PROGRAM PRG_SL2K0_POWER
VAR
    {attribute 'pytmc' := '
        pv: SL2K0:POWER
        io: io
    '}
    {attribute 'TcLinkTo' := '.RTD_South_1.iRaw := TIIB[SL2K0-EL3202-E8]^RTD Inputs Channel 1^Value;
                              .RTD_South_1.bError := TIIB[SL2K0-EL3202-E8]^RTD Inputs Channel 1^Status^Error;
                              .RTD_South_1.bUnderrange := TIIB[SL2K0-EL3202-E8]^RTD Inputs Channel 1^Status^Underrange;
                              .RTD_South_1.bOverrange := TIIB[SL2K0-EL3202-E8]^RTD Inputs Channel 1^Status^Overrange;
                              .RTD_South_2.iRaw := TIIB[SL2K0-EL3202-E8]^RTD Inputs Channel 2^Value;
                              .RTD_South_2.bError := TIIB[SL2K0-EL3202-E8]^RTD Inputs Channel 2^Status^Error;
                              .RTD_South_2.bUnderrange := TIIB[SL2K0-EL3202-E8]^RTD Inputs Channel 2^Status^Underrange;
                              .RTD_South_2.bOverrange := TIIB[SL2K0-EL3202-E8]^RTD Inputs Channel 2^Status^Overrange;
                              .RTD_TOP_1.iRaw := TIIB[SL2K0-EL3202-E9]^RTD Inputs Channel 1^Value;
                              .RTD_TOP_1.bError := TIIB[SL2K0-EL3202-E9]^RTD Inputs Channel 1^Status^Error;
                              .RTD_TOP_1.bUnderrange := TIIB[SL2K0-EL3202-E9]^RTD Inputs Channel 1^Status^Underrange;
                              .RTD_TOP_1.bOverrange := TIIB[SL2K0-EL3202-E9]^RTD Inputs Channel 1^Status^Overrange;
                              .RTD_TOP_2.iRaw := TIIB[SL2K0-EL3202-E9]^RTD Inputs Channel 2^Value;
                              .RTD_TOP_2.bError := TIIB[SL2K0-EL3202-E9]^RTD Inputs Channel 2^Status^Error;
                              .RTD_TOP_2.bUnderrange := TIIB[SL2K0-EL3202-E9]^RTD Inputs Channel 2^Status^Underrange;
                              .RTD_TOP_2.bOverrange := TIIB[SL2K0-EL3202-E9]^RTD Inputs Channel 2^Status^Overrange;
                              .RTD_North_1.iRaw := TIIB[SL2K0-EL3202-E10]^RTD Inputs Channel 1^Value;
                              .RTD_North_1.bError := TIIB[SL2K0-EL3202-E10]^RTD Inputs Channel 1^Status^Error;
                              .RTD_North_1.bUnderrange := TIIB[SL2K0-EL3202-E10]^RTD Inputs Channel 1^Status^Underrange;
                              .RTD_North_1.bOverrange := TIIB[SL2K0-EL3202-E10]^RTD Inputs Channel 1^Status^Overrange;
                              .RTD_North_2.iRaw := TIIB[SL2K0-EL3202-E10]^RTD Inputs Channel 2^Value;
                              .RTD_North_2.bError := TIIB[SL2K0-EL3202-E10]^RTD Inputs Channel 2^Status^Error;
                              .RTD_North_2.bUnderrange := TIIB[SL2K0-EL3202-E10]^RTD Inputs Channel 2^Status^Underrange;
                              .RTD_North_2.bOverrange := TIIB[SL2K0-EL3202-E10]^RTD Inputs Channel 2^Status^Overrange;
                              .RTD_Bottom_1.iRaw := TIIB[SL2K0-EL3202-E10]^RTD Inputs Channel 1^Value;
                              .RTD_Bottom_1.bError := TIIB[SL2K0-EL3202-E10]^RTD Inputs Channel 1^Status^Error;
                              .RTD_Bottom_1.bUnderrange := TIIB[SL2K0-EL3202-E11]^RTD Inputs Channel 1^Status^Underrange;
                              .RTD_Bottom_1.bOverrange := TIIB[SL2K0-EL3202-E11]^RTD Inputs Channel 1^Status^Overrange;
                              .RTD_Bottom_2.iRaw := TIIB[SL2K0-EL3202-E11]^RTD Inputs Channel 2^Value;
                              .RTD_Bottom_2.bError := TIIB[SL2K0-EL3202-E11]^RTD Inputs Channel 2^Status^Error;
                              .RTD_Bottom_2.bUnderrange := TIIB[SL2K0-EL3202-E11]^RTD Inputs Channel 2^Status^Underrange;
                              .RTD_Bottom_2.bOverrange := TIIB[SL2K0-EL3202-E11]^RTD Inputs Channel 2^Status^Overrange'}
    fbSL2K0: FB_SLITS_POWER;
//GET PMP Move Ok bit
// Default True until it is properly linked to PMPS bit
    bMoveOk:BOOL :=TRUE;
    {attribute 'pytmc' := '
    pv: SL2K0:POWER:GO;
    io: io;
    field: ZNAM False;
    field: ONAM True;
    '}
    bExecuteMotion:BOOL ;
    //for testing purposes only. comment-out/delete once done.
    mcPower : ARRAY [1..4] OF MC_POWER;
END_VAR


fbSL2K0.bMoveOk := bMoveOk;

fbSL2K0(stTopBlade:=  Main.M22,
        stBottomBlade:= Main.M23,
        stNorthBlade:=  Main.M24,
        stSouthBlade:=  Main.M25,
        bExecuteMotion:=bExecuteMotion);


//for testing purposes only. comment-out/delete once done.
(*mcPower[1](axis:=Main.M22.Axis, Enable:=TRUE, enable_positive:=Main.M22.bLimitForwardEnable, enable_negative:=Main.M22.bLimitBackwardEnable);
mcPower[2](axis:=Main.M23.Axis, Enable:=TRUE, enable_positive:=Main.M23.bLimitForwardEnable, enable_negative:=Main.M23.bLimitBackwardEnable);
mcPower[3](axis:=Main.M24.Axis, Enable:=TRUE, enable_positive:=Main.M24.bLimitForwardEnable, enable_negative:=Main.M24.bLimitBackwardEnable);
mcPower[4](axis:=Main.M25.Axis, Enable:=TRUE, enable_positive:=Main.M25.bLimitForwardEnable, enable_negative:=Main.M25.bLimitBackwardEnable);*)

END_PROGRAM

(* stored: Version 1.1.0.1, ProductVersion 3.1.4022.18
   POU PRG_SL2K0_POWER: Id {c8e49e09-7b9e-4d82-ac5a-e310bf9e41e1}, SpecialFunc None *)
